Universal Robots PolyScope program: mt_rtde_control_loop.urp

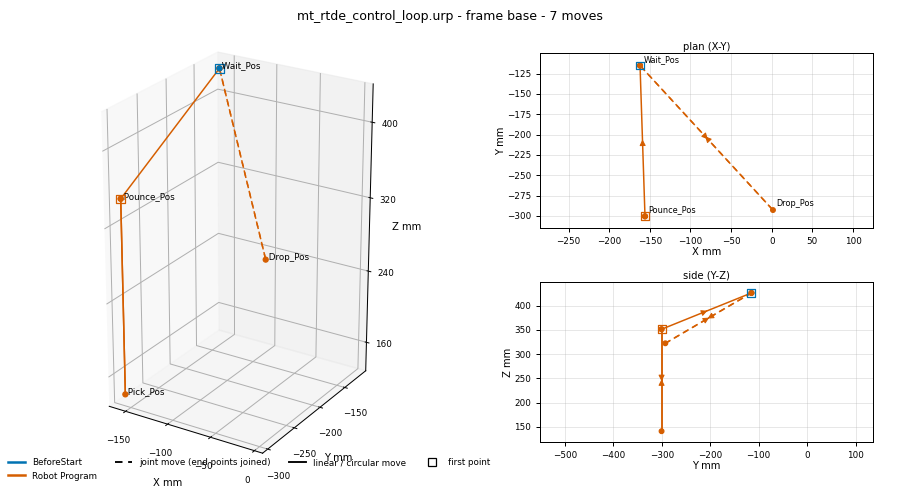
[picture p0: tool path of mt_rtde_control_loop.urp in frame base, 7 of 7 moves have a stored position in this frame; points joined in program order, loops and branches not executed]
Program mt_rtde_control_loop (installation=default directory=/home/ur/ursim-current/programs createdIn=3.2.19275 lastSavedIn=5.14.5 robotSerialNumber=20195399999)
Calibrated DH parameters: a=[0, -0.24355, -0.2132, 0, 0, 0]; d=[0.15185, 0, 0, 0.13105, 0.08535, 0.0921]; alpha=[1.570796, 0, 0, 1.570796, -1.570796, 0]; deltaTheta=[0, 0, 0, 0, 0, 0]
InitVariablesNode variables(variable(name=COBOT_IDLE, expression=1), variable(name=COBOT_INIT, expression=0), variable(name=COBOT_PICKING, expression=2), variable(name=PRINTER_IDLE, expression=1), variable(name=PRINTER_RUNNING, expression=2))
BeforeStart
  PRINTER_IDLE := 1
  PRINTER_RUNNING := 2
  COBOT_INIT := 0
  COBOT_IDLE := 1
  COBOT_PICKING := 2
  MoveJ speed 60 deg/s, acceleration 80 deg/s^2 (useActiveTCP=true) feature=Plane_1
    Waypoint Wait_Pos: TCP in base x=-162.083 y=-115.036 z=426.33 mm, rx=-0.2156 ry=3.1342 rz=0 rad; joints [-103.385, -67.105, -71.055, -131.84, 90, -21.256] deg; feature pose in base x=-207.753 y=-250.403 z=219.284 mm, rx=0 ry=0 rz=2.9224 rad
  Set DigitalOutput pin=tool_out[0]; digitalValue=0
  Script: rtde_set_watchdog("input_int_register_0", 1, "PAUSE")
  Script: write_output_integer_register(0, COBOT_INIT)
Robot Program (runOnlyOnce=false)
  Wait Condition expression=read_input_integer_register(0)≟PRINTER_IDLE
  'Ready to remove item from print bed'
  Script: write_output_integer_register(0,COBOT_PICKING)
  Folder Pick and Deposit
    MoveL speed 250 mm/s, acceleration 1200 mm/s^2 (useActiveTCP=true) feature=Plane_1
      Waypoint Pounce_Pos: TCP in base x=-155.983 y=-300.636 z=351.33 mm, rx=-0.2156 ry=3.1342 rz=0 rad; joints [-94.659, -103.78, -38.635, -127.585, 90, -12.53] deg; TCP offset x=0 y=0 z=75 mm, rx=0 ry=0 rz=0 rad; feature pose in base x=-207.753 y=-250.403 z=219.284 mm, rx=0 ry=0 rz=2.9224 rad
    'Make sure grabber is open'
    MoveL speed 250 mm/s, acceleration 1200 mm/s^2 (useActiveTCP=true) feature=Plane_1
      Waypoint Pick_Pos: TCP in base x=-155.983 y=-300.636 z=140.787 mm, rx=-0.2156 ry=3.1342 rz=0 rad; joints [-94.659, -97.463, -106.165, -66.372, 90, -12.53] deg
    'Close grabber'
    Set DigitalOutput pin=tool_out[0]; digitalValue=1
    Wait Sleep waitTime=0.25
    SetPayload (workpieceName=Load)
    MoveL speed 250 mm/s, acceleration 1200 mm/s^2 (useActiveTCP=true) feature=Plane_1
      Waypoint Pounce_Pos: TCP in base x=-155.983 y=-300.636 z=351.33 mm, rx=-0.2156 ry=3.1342 rz=0 rad; joints [-94.659, -103.78, -38.635, -127.585, 90, -12.53] deg
      Waypoint Wait_Pos: TCP in base x=-162.083 y=-115.036 z=426.33 mm, rx=-0.2156 ry=3.1342 rz=0 rad; joints [-103.385, -67.105, -71.055, -131.84, 90, -21.256] deg; feature pose in base x=-207.753 y=-250.403 z=219.284 mm, rx=0 ry=0 rz=2.9224 rad
    MoveJ speed 60 deg/s, acceleration 80 deg/s^2 (useActiveTCP=true) feature=Plane_1
      Waypoint Drop_Pos: TCP in base x=1.49 y=-292.872 z=322.341 mm, rx=-1.2325 ry=2.8897 rz=0 rad; joints [-63.128, -81.612, -92.561, -95.827, 90, -19.327] deg; feature pose in base x=-207.753 y=-250.403 z=219.284 mm, rx=0 ry=0 rz=2.9224 rad
    'Drop Item'
    Set DigitalOutput pin=tool_out[0]; digitalValue=0
    Wait Sleep waitTime=0.25
    SetPayload (workpieceName=No_Load)
    MoveJ speed 60 deg/s, acceleration 80 deg/s^2 (useActiveTCP=true) feature=Plane_1
      Waypoint Wait_Pos: TCP in base x=-162.083 y=-115.036 z=426.33 mm, rx=-0.2156 ry=3.1342 rz=0 rad; joints [-103.385, -67.105, -71.055, -131.84, 90, -21.256] deg; feature pose in base x=-207.753 y=-250.403 z=219.284 mm, rx=0 ry=0 rz=2.9224 rad
  'Confirm pick and drop was completed'
  Script: write_output_integer_register(0,COBOT_IDLE)
  'Wait Until Client Controller Acknowledges Confirmation'
  Wait Condition expression=read_input_integer_register(0)≟PRINTER_RUNNING
  Script: sync()
